TYPE TcSymbolInfo :
STRUCT
	nAddress	: UDINT; 
	nLength		: UDINT; 
END_STRUCT
END_TYPE

(* stored: Version 1.1.0.1, ProductVersion 3.1.4022.6
   DUT TcSymbolInfo: Id {53ac5aaa-067c-44ff-891e-de8a3402f5af} *)
